// TIA Portal V17 export
// export: Created 2024-09-02T12:50:16.5763703Z, ExportSetting WithDefaults, DisplayName Totally Integrated Automation Portal, DisplayVersion V17, DisplayName TIA Portal Openness, DisplayVersion V17, DisplayName TIA Portal Version Control Interface, DisplayVersion V17, DisplayName STEP 7 Professional, DisplayVersion V17, DisplayName STEP 7 Safety, DisplayVersion V17, DisplayName WinCC Professional, DisplayVersion V17
DATA_BLOCK "AnwDB_Door_OP70"   // DB149
{ S7_Optimized_Access := 'TRUE'; DB_Accessible_From_OPC_UA := 'FALSE' }
AUTHOR : VAF
FAMILY : SG
NAME : SG
VERSION : 0.1
// stored: AutoNumber true, DBAccessibleFromOPCUA false, IsOnlyStoredInLoadMemory false, IsRetainMemResEnabled false, IsWriteProtectedInAS false, MemoryReserve 0
   VAR
      Geleral : Struct
         ACK { ExternalWritable := 'False'} : Bool;   // Fehler quittieren / Acknowledge error
         Stop_at_endOfCycle : Bool;   // Halt nach Taktende von Schutztürtaster / Stop after end of cycle of safety door pushbutton
      END_STRUCT;
      Button_HP : Struct   // Hauptpult gilt für alle Schutztüren / Main console applies to all safety doors
         Door_Open : Bool;   // Schutztür öffnen / Protective door open
         Door_Close : Bool;   // Schutztür schliessen / Close safety door
         Req_Door_Open : Bool;   // Anforderung Schutztür öffnen / Requirement of Safety Door opened
      END_STRUCT;
      SG1 { S7_SetPoint := 'True'} : "TypeSafetyDoor";   // Schutztür Station / Safety door Station
      SG2 { S7_SetPoint := 'True'} : "TypeSafetyDoor";   // Schutztür Drucker / Protective door Printer
      SG3 { S7_SetPoint := 'True'} : "TypeSafetyDoor";   // Schutztür xxx / Safety door XXX
      SG4 { S7_SetPoint := 'True'} : "TypeSafetyDoor";   // Schutztür xxx / Safety door XXX
   END_VAR
BEGIN
END_DATA_BLOCK
